{attribute 'linkalways'}
{attribute 'hide_all_locals'}
FUNCTION_BLOCK ValueDword EXTENDS ValueDwordRead IMPLEMENTS Value
VAR
END_VAR

METHOD SetFromType : BOOL
VAR_INPUT
	source : __SYSTEM.AnyType;
END_VAR
SetFromType := ConvertAnyType(source, thisAnyType);
END_METHOD

METHOD SetFromString : BOOL
VAR_INPUT
	value : T_MaxString;
END_VAR
thisValue := STRING_TO_DWORD(value);

SetFromString := TRUE;
END_METHOD

METHOD Set : BOOL
VAR_INPUT
	source : ANY;
END_VAR
Set := ConvertAnyType(source, thisAnyType);
END_METHOD

END_FUNCTION_BLOCK

(* stored: Version 1.1.0.1
   POU ValueDword: Id {940ced1a-330e-4e15-bcd1-d98f14813c5b}, SpecialFunc None
   Method SetFromType: Id {a3b81139-aea0-4829-8fae-1ea1a0eefbff}
   Method SetFromString: Id {682d523e-f885-485d-a76e-4b2a6f434650}
   Method Set: Id {a152ed86-0cbf-4eb5-b1ac-34ea9b1a7b20} *)
